// TIA Portal project "guvenlik_cpu" (V18)

(* hardware
DEVICE "S7-1200 station_1"  S7-1200 Station
   slot 0: "Rack_0"  S7-1200 Rack  Rack  V1.0
   slot 1: "PLC_1"  CPU 1214FC DC/DC/DC  6ES7 214-1AF40-0XB0  V4.6
DEVICE "ET 200S station_1"  ET 200S station
   slot 0: "Rack_0"  Rail
   slot 0: "IO device_1"  IM 151-3 PN ST  6ES7 151-3AA22-0AB0  V5.0
   slot 1: "PM-E 24VDC_1"  PM-E 24VDC  6ES7 138-4CA01-0AA0
   slot 2: "4/8 F-DI DC24V_1"  4/8 F-DI DC24V  6ES7 138-4FA03-0AB0
   slot 3: "4 F-DO DC24V/2A_1"  4 F-DO DC24V/2A  6ES7 138-4FB02-0AB0
*)

// ===== PLC "PLC_1"  CPU 1214FC DC/DC/DC =====

DATA_BLOCK "Main_Safety_RTG1_DB"   // DB1, F_DB
{ S7_Optimized_Access := 'TRUE' }
NAME : FUSI
VERSION : 0.1
// stored: InstanceOfName Main_Safety_RTG1
"Main_Safety_RTG1"
BEGIN
END_DATA_BLOCK

FUNCTION_BLOCK "Main_Safety_RTG1"   // FB1, F_FBD
{ S7_Optimized_Access := 'TRUE' }
BEGIN
END_FUNCTION_BLOCK

ORGANIZATION_BLOCK "Main"   // OB1, LAD, ProgramCycle
TITLE = "Main Program Sweep (Cycle)"
{ S7_Optimized_Access := 'TRUE' }
VERSION : 0.1
   VAR_INPUT
      Initial_Call : Bool;   // Initial call of this OB
      Remanence : Bool;   // =True, if remanent data are available
   END_VAR
BEGIN
END_ORGANIZATION_BLOCK